MoveJ RelTool (starting_position, 72,-16, -535.4 \Rx:=8, \Ry:=-2.1, \Rz:=-4), v200, z200, Tooldata_9;
MoveJ RelTool (starting_position, 73,-16, -534.8 \Rx:=8.2, \Ry:=-2.1, \Rz:=-4), v200, z200, Tooldata_9;
MoveJ RelTool (starting_position, 74,-16, -534.4 \Rx:=8.4, \Ry:=-2.1, \Rz:=-4), v200, z200, Tooldata_9;
MoveJ RelTool (starting_position, 75,-16, -534.1 \Rx:=8.5, \Ry:=-1.8, \Rz:=-4), v200, z200, Tooldata_9;
MoveJ RelTool (starting_position, 76,-16, -534 \Rx:=8.7, \Ry:=-1.8, \Rz:=-4), v200, z200, Tooldata_9;
MoveJ RelTool (starting_position, 77,-16, -533.8 \Rx:=8.8, \Ry:=-1.5, \Rz:=-4), v200, z200, Tooldata_9;
MoveJ RelTool (starting_position, 79,-16, -533.5 \Rx:=9, \Ry:=-1.5, \Rz:=-4), v200, z200, Tooldata_9;
MoveJ RelTool (starting_position, 81,-16, -533.1 \Rx:=9.1, \Ry:=-1.2, \Rz:=-4), v200, z200, Tooldata_9;
MoveJ RelTool (starting_position, 83,-16, -532.4 \Rx:=9.3, \Ry:=-1.2, \Rz:=-4), v200, z200, Tooldata_9;
MoveJ RelTool (starting_position, 85,-16, -531.4 \Rx:=9.4, \Ry:=-0.9, \Rz:=-4), v200, z200, Tooldata_9;
MoveJ RelTool (starting_position, 87,-16, -530 \Rx:=9.6, \Ry:=-0.6, \Rz:=-4), v200, z200, Tooldata_9;
MoveJ RelTool (starting_position, 89,-20, -528.5 \Rx:=9.7, \Ry:=-0.6, \Rz:=-5), v200, z200, Tooldata_9;
MoveJ RelTool (starting_position, 92,-20, -526.8 \Rx:=9.8, \Ry:=-0.3, \Rz:=-5), v200, z200, Tooldata_9;
MoveJ RelTool (starting_position, 94,-20, -525.2 \Rx:=10, \Ry:=-0, \Rz:=-5), v200, z200, Tooldata_9;
MoveJ RelTool (starting_position, 96,-20, -523.7 \Rx:=10.1, \Ry:=0, \Rz:=-5), v200, z200, Tooldata_9;
MoveJ RelTool (starting_position, 99,-20, -522.4 \Rx:=10.2, \Ry:=0.3, \Rz:=-5), v200, z200, Tooldata_9;
MoveJ RelTool (starting_position, 101,-20, -521.5 \Rx:=10.4, \Ry:=0.6, \Rz:=-5), v200, z200, Tooldata_9;
MoveJ RelTool (starting_position, 104,-20, -520.9 \Rx:=10.5, \Ry:=0.9, \Rz:=-5), v200, z200, Tooldata_9;
MoveJ RelTool (starting_position, 106,-20, -520.5 \Rx:=10.6, \Ry:=0.9, \Rz:=-5), v200, z200, Tooldata_9;
MoveJ RelTool (starting_position, 109,-20, -520.5 \Rx:=10.7, \Ry:=1.2, \Rz:=-5), v200, z200, Tooldata_9;
MoveJ RelTool (starting_position, 111,-20, -520.8 \Rx:=10.9, \Ry:=1.5, \Rz:=-5), v200, z200, Tooldata_9;
MoveJ RelTool (starting_position, 114,-20, -521.4 \Rx:=11, \Ry:=1.8, \Rz:=-5), v200, z200, Tooldata_9;
MoveJ RelTool (starting_position, 116,-20, -522.3 \Rx:=11.1, \Ry:=2.1, \Rz:=-5), v200, z200, Tooldata_9;
MoveJ RelTool (starting_position, 118,-20, -523.5 \Rx:=11.2, \Ry:=2.1, \Rz:=-5), v200, z200, Tooldata_9;
MoveJ RelTool (starting_position, 119,-20, -525 \Rx:=11.3, \Ry:=2.4, \Rz:=-5), v200, z200, Tooldata_9;
MoveJ RelTool (starting_position, 121,-24, -526.8 \Rx:=11.4, \Ry:=2.4, \Rz:=-6), v200, z200, Tooldata_9;
MoveJ RelTool (starting_position, 122,-24, -528.8 \Rx:=11.5, \Ry:=2.4, \Rz:=-6), v200, z200, Tooldata_9;
MoveJ RelTool (starting_position, 123,-24, -531 \Rx:=11.6, \Ry:=2.7, \Rz:=-6), v200, z200, Tooldata_9;
MoveJ RelTool (starting_position, 123,-24, -533.4 \Rx:=11.8, \Ry:=2.7, \Rz:=-6), v200, z200, Tooldata_9;
MoveJ RelTool (starting_position, 124,-24, -535.9 \Rx:=11.8, \Ry:=2.7, \Rz:=-6), v200, z200, Tooldata_9;
MoveJ RelTool (starting_position, 124,-24, -538.6 \Rx:=11.9, \Ry:=2.7, \Rz:=-6), v200, z200, Tooldata_9;
MoveJ RelTool (starting_position, 123,-24, -541.4 \Rx:=12, \Ry:=2.7, \Rz:=-6), v200, z200, Tooldata_9;
MoveJ RelTool (starting_position, 122,-24, -544.3 \Rx:=12.1, \Ry:=2.7, \Rz:=-6), v200, z200, Tooldata_9;
MoveJ RelTool (starting_position, 121,-24, -547.1 \Rx:=12.2, \Ry:=2.4, \Rz:=-6), v200, z200, Tooldata_9;
MoveJ RelTool (starting_position, 120,-24, -549.8 \Rx:=12.3, \Ry:=2.4, \Rz:=-6), v200, z200, Tooldata_9;
MoveJ RelTool (starting_position, 119,-24, -552.3 \Rx:=12.4, \Ry:=2.1, \Rz:=-6), v200, z200, Tooldata_9;
MoveJ RelTool (starting_position, 117,-24, -554.4 \Rx:=12.5, \Ry:=2.1, \Rz:=-6), v200, z200, Tooldata_9;
MoveJ RelTool (starting_position, 115,-24, -556 \Rx:=12.5, \Ry:=1.8, \Rz:=-6), v200, z200, Tooldata_9;
MoveJ RelTool (starting_position, 113,-24, -557.3 \Rx:=12.6, \Ry:=1.8, \Rz:=-6), v200, z200, Tooldata_9;
MoveJ RelTool (starting_position, 110,-24, -558.3 \Rx:=12.7, \Ry:=1.5, \Rz:=-6), v200, z200, Tooldata_9;
MoveJ RelTool (starting_position, 107,-24, -558.9 \Rx:=12.8, \Ry:=1.2, \Rz:=-6), v200, z200, Tooldata_9;
MoveJ RelTool (starting_position, 105,-28, -559.3 \Rx:=12.8, \Ry:=0.9, \Rz:=-7), v200, z200, Tooldata_9;
MoveJ RelTool (starting_position, 102,-28, -559.6 \Rx:=12.9, \Ry:=0.6, \Rz:=-7), v200, z200, Tooldata_9;
MoveJ RelTool (starting_position, 99,-28, -559.7 \Rx:=12.9, \Ry:=0.3, \Rz:=-7), v200, z200, Tooldata_9;
MoveJ RelTool (starting_position, 95,-28, -559.7 \Rx:=13, \Ry:=0, \Rz:=-7), v200, z200, Tooldata_9;
MoveJ RelTool (starting_position, 92,-28, -559.5 \Rx:=13.1, \Ry:=-0, \Rz:=-7), v200, z200, Tooldata_9;
MoveJ RelTool (starting_position, 89,-28, -559.2 \Rx:=13.1, \Ry:=-0.3, \Rz:=-7), v200, z200, Tooldata_9;
MoveJ RelTool (starting_position, 86,-28, -558.6 \Rx:=13.2, \Ry:=-0.9, \Rz:=-7), v200, z200, Tooldata_9;
MoveJ RelTool (starting_position, 83,-28, -557.8 \Rx:=13.2, \Ry:=-1.2, \Rz:=-7), v200, z200, Tooldata_9;
MoveJ RelTool (starting_position, 80,-28, -556.5 \Rx:=13.3, \Ry:=-1.5, \Rz:=-7), v200, z200, Tooldata_9;
MoveJ RelTool (starting_position, 77,-28, -554.7 \Rx:=13.3, \Ry:=-1.8, \Rz:=-7), v200, z200, Tooldata_9;
MoveJ RelTool (starting_position, 74,-28, -552.6 \Rx:=13.3, \Ry:=-1.8, \Rz:=-7), v200, z200, Tooldata_9;
MoveJ RelTool (starting_position, 71,-28, -550 \Rx:=13.4, \Ry:=-2.1, \Rz:=-7), v200, z200, Tooldata_9;
MoveJ RelTool (starting_position, 68,-28, -547.1 \Rx:=13.4, \Ry:=-2.4, \Rz:=-7), v200, z200, Tooldata_9;
MoveJ RelTool (starting_position, 66,-28, -544.1 \Rx:=13.5, \Ry:=-2.7, \Rz:=-7), v200, z200, Tooldata_9;
MoveJ RelTool (starting_position, 63,-28, -541 \Rx:=13.5, \Ry:=-2.7, \Rz:=-7), v200, z200, Tooldata_9;
MoveJ RelTool (starting_position, 61,-28, -538.1 \Rx:=13.5, \Ry:=-3, \Rz:=-7), v200, z200, Tooldata_9;
MoveJ RelTool (starting_position, 59,-28, -535.7 \Rx:=13.6, \Ry:=-3.3, \Rz:=-7), v200, z200, Tooldata_9;
MoveJ RelTool (starting_position, 57,-28, -533.7 \Rx:=13.6, \Ry:=-3.3, \Rz:=-7), v200, z200, Tooldata_9;
MoveJ RelTool (starting_position, 56,-28, -532.2 \Rx:=13.6, \Ry:=-3.6, \Rz:=-7), v200, z200, Tooldata_9;
MoveJ RelTool (starting_position, 55,-28, -531.2 \Rx:=13.6, \Ry:=-3.6, \Rz:=-7), v200, z200, Tooldata_9;
MoveJ RelTool (starting_position, 53,-28, -530.8 \Rx:=13.6, \Ry:=-3.9, \Rz:=-7), v200, z200, Tooldata_9;
MoveJ RelTool (starting_position, 52,-28, -530.6 \Rx:=13.6, \Ry:=-3.9, \Rz:=-7), v200, z200, Tooldata_9;
MoveJ RelTool (starting_position, 52,-28, -530.8 \Rx:=13.6, \Ry:=-3.9, \Rz:=-7), v200, z200, Tooldata_9;
MoveJ RelTool (starting_position, 51,-28, -531.1 \Rx:=13.7, \Ry:=-4.2, \Rz:=-7), v200, z200, Tooldata_9;









    ENDPROC

! function used to produce movement
    PROC move(num x, num z,num rx, num ry, num rz, num joint1)
     ConfJ\On;

     !!!! Method Two !!!!!!
     !current_position :=RelTool(CRobT(\TaskName:="T_ROB1"\Tool:=Tooldata_9), x,0, z \Rx:=rx, \Ry:=ry, \Rz:=0);
     !joints := CalcJointT(current_position,Tooldata_9 \WObj:=wobj0);
    ! joints.robax.rax_1 :=joint1;
     !MoveAbsJ joints,v200,z10,Tooldata_9,\WObj:=wobj0;
     !!!!!!!!!!!!!!!!!!!!!!!!!!!!!

     MoveJ RelTool(starting_position, x,0, z \Rx:=rx, \Ry:=ry, \Rz:=rz),v200,z200,Tooldata_9;



     !!!!! Method One !!!!!!
    ! MoveJ (RelTool (CRobT(\TaskName:="T_ROB1"\Tool:=Tooldata_9), x,0, z \Rx:=rx, \Ry:=ry, \Rz:=0)),v200,z200,Tooldata_9;
    !joints := CJointT(\TaskName:="T_ROB1");
    !joints.robax.rax_1 := joint1;
    ! MoveAbsJ joints,v200,fine,Tooldata_9,\WObj:=wobj0;
    !!!!!!!!!!!!!!!!!!!!!!!!!!!!!!!!!!!!!!!
    ENDPROC



ENDMODULE
